Staubli VAL3: onRun.pgx

public program onRun(string& x_sItem[] (dimensions=1))
begin
  // PROG NAME x_sItem
  // SET THE CALL SUB..
  cycleStatus:bCALL=true
  if x_sItem!=""
    cycleStatus:iToSuperV.sType="PROG"
    cycleStatus:iToSuperV.sData=x_sItem
  endIf
  use:bUseRefresh=true
end
